// TwinCAT 3 PLC project MimoControl
// ProgramVersion: 3.1.4023.0
// libraries:
//   Tc2_ControllerToolbox,3.4.1.4,Beckhoff Automation GmbH
//   Tc2_Math,3.3.1.0,Beckhoff Automation GmbH
//   Tc2_Standard,3.3.3.0,Beckhoff Automation GmbH
//   Tc2_System,3.4.22.0,Beckhoff Automation GmbH
//   Tc2_TempController,3.3.4.0,Beckhoff Automation GmbH
//   Tc3_Module,3.3.21.0,Beckhoff Automation GmbH
// project tree:
//   GVLs/ gbl.TcGVL
//   / PlcTask.TcTTO (not stored)
//   POUs/ MAIN.TcPOU (not stored)
// real-time tasks:
//   TASK PlcTask: cycle T#10ms, priority 20, ADS port 350

// ---- GVLs/gbl.TcGVL
{attribute 'qualified_only'}
VAR_GLOBAL
	bRampingEnable : BOOL;	

	fRampingValue:LREAL; 
	fTargetTemp : LREAL;
	
	fSetManual					:			LREAL;	
	eCTRL_MODE	: E_CTRL_MODE;
	bStart:BOOL;
	P_Value:ARRAY[1..4] OF LREAL:= [3, 3, 3, 3];
	I_Value:ARRAY[1..4] OF TIME:= [T#5S, T#5S, T#5S, T#5S];
	D_Value:ARRAY[1..4] OF TIME:= [T#50S, T#50S, T#50S, T#50S];
	fPowerLimit:REAL;
	
END_VAR
